{attribute 'linkalways'} 
{attribute 'no_explicit_call' := 'This FB is a CLASS and must be accessed using methods or properties'}
{attribute 'enable_dynamic_creation'}
FUNCTION_BLOCK _PVOID EXTENDS DatatypeBase
VAR
	localData : PVOID;
	activeData : REFERENCE TO PVOID REF= localData;
END_VAR

PROPERTY PUBLIC Address : PVOID
GET
Address := ADR(activeData);
END_GET
END_PROPERTY

METHOD PUBLIC ClearReference
VAR_INPUT
END_VAR
activeData REF= localData;
END_METHOD

METHOD PUBLIC Clone : I_Datatype
VAR
    pClone : POINTER TO _PVOID;
END_VAR
pClone := __NEW(_PVOID);
Clone := pClone^;
END_METHOD

METHOD PUBLIC MakeReferenceTo
VAR_INPUT
	ReferenceTarget : REFERENCE TO PVOID;
END_VAR
activeData REF= ReferenceTarget;
END_METHOD

METHOD PUBLIC SerializeWith
VAR_INPUT
	Serializer : I_Serializer;
END_VAR
VAR
	pVoidAsString : T_MAXSTRING;
END_VAR
pVoidAsString := pvoid_To_string(activeData);
Serializer.AddString(pVoidAsString);
END_METHOD

PROPERTY PUBLIC Size : UDINT
GET
Size := SIZEOF(activeData);
END_GET
END_PROPERTY

METHOD TryDeserializeFrom : BOOL
VAR_INPUT
	Deserializer : I_Deserializer;
	Feedback : I_DeserializerFeedback;
END_VAR
VAR
	pVoidAsString : T_MAXSTRING;
END_VAR
IF NOT Deserializer.TryGetString(pVoidAsString, Feedback) THEN
	RETURN;
END_IF

activeData := STRING_TO_PVOID(pVoidAsString);
TryDeserializeFrom := TRUE;
END_METHOD

METHOD TryMakeReferenceTo : BOOL
VAR_INPUT
	Target : I_Datatype;
END_VAR
VAR
	pTargetData : POINTER TO PVOID;
END_VAR
IF NOT IsEquivalentTo(Target) THEN
	RETURN;
END_IF

pTargetData := Target.Address;
activeData REF= pTargetData^;
TryMakeReferenceTo := TRUE;
END_METHOD

PROPERTY PUBLIC TypeName : T_MAXSTRING
GET
TypeName := 'PVOID';
END_GET
END_PROPERTY

PROPERTY PUBLIC Value : REFERENCE TO PVOID
GET
Value REF= activeData;
END_GET
END_PROPERTY

END_FUNCTION_BLOCK

(* stored: Version 1.1.0.1, ProductVersion 3.1.4024.13
   POU _PVOID: Id {ece32e5e-6487-0057-3c19-512c10e5e626}, SpecialFunc None
   Property Address: Id {71578cee-4238-0958-1a38-1d8a71280df4}
   Get Get: Id {191a49cb-ac08-06fd-14cd-5a2c0d5ff2a2}
   Method ClearReference: Id {2f14f86a-6104-0063-361e-9a07da8ca1d2}
   Method Clone: Id {b5eb3fa2-14c6-0e04-09a7-b6439e43fc81}
   Method MakeReferenceTo: Id {472f3e7d-7bf3-05d9-0466-aa215d041bc6}
   Method SerializeWith: Id {de58bb39-1d4a-0e23-2c2c-e4bf80b9c178}
   Property Size: Id {5e312ff8-84f0-0b61-0f4d-ad09d4501058}
   Get Get: Id {535be1f1-8391-066d-1834-a29d2cd94d16}
   Method TryDeserializeFrom: Id {45b86e97-9769-06db-21a4-8a58cb8cc6b2}
   Method TryMakeReferenceTo: Id {1b5ed480-f958-060c-2931-5e4fee2f1b78}
   Property TypeName: Id {2f0de6b3-5434-090f-3be7-268c1a830974}
   Get Get: Id {4a16a719-7c0a-0d39-3387-0a3efb294a7a}
   Property Value: Id {4559dc0b-2c04-0410-0c6b-dfa3fe90cee5}
   Get Get: Id {2fde5ab5-7258-087a-1af2-47ade5c7b474} *)
